(* Schneider Machine Expert - Basic project Grease Machine, file version 2.6.0.0 *)
(* ProjectInformations: Name=New project *)

HARDWARE
  Cpu 0: TM221CE40R
  EthernetConfiguration: NetworkName=M221, IpAllocationMode=FixedAddress, IpAddress=192.168.0.3, SubnetMask=255.255.255.0
  SerialLineConfiguration: Baud=Baud19200, Parity=ParityEven, DataBits=DataBits8, StopBits=StopBits1, PhysicalMedium=PhysicalMediumRs485, TransmissionMode=TransmissionModeModbusRtu, SlaveId=1, Addressing=SlaveAddressing
  MastTask: UsePeriodScanMode=false, PeriodScan=100
  FastTask: Period=255
  CpuBehavior: StartingMode=StartAsPreviousState, AutoSaveRamOnEeprom=true, WatchdogPeriod=250

SYMBOLS  (address, symbol, comment, settings)
  %M0         "RST HMI"
  %M1         "M_BTN START"
  %M2         "M_SENSOR CERTAIN"
  %M3         "M_SENSOR TABLE"
  %M4         "M_BTN CYCLE START"
  %M5         "M_EMG"
  %M6         "M_PROCESS DONE"
  %M7         "M_GREASE EMPTY"
  %M8         "M_GREASE TRIGGER"
  %M9         "M_Q GREASE ACTIVE"
  %M10        "M_Q CERTAIN SENSOR"
  %M11        "M_Q CYCLE START"
  %M12        "M_Q EMERGENCY"
  %M13        "M_Q RED LAMP"
  %M14        "M_Q YELLOW LAMP"
  %M15        "M_Q GREEN LAMP"
  %M16        "M_Q BUZZER"
  %M17        "RED LAMP 2"
  %M18        "TRIGGER YELLOW LAMP"
  %M19        "PAUSE"
  %M20        "FINISH RUN"
  %M21        "RESET BUZZER"
  %M22        "MEMORY M2"
  %M23        "M_TABLE_HMI"
  %M30        "M_START"
  %M31        "M_START HMI"
  %M32        "M_RUN_EMG"
  %M33        "TRIGER_ROBOT_HOME"
  %M34        "ROBOT_GO_HOME"
  %M47        "M_EMG"
  %M49        "POLARITY CHECKED"
  %M50        "NEGATIVE"
  %M51        "POSITIVE"
  %M52        "FIRST RUN"
  %M53        "DONE CUTTING"
  %M54        "NEGATIVE READY"
  %M55        "TRIGGER"
  %M56        "COUNTER OUTPUT"
  %M100       "START GUI"
  %M102       "M_START"
  %MW0        "Count Output"
  %I0.1       "BTN START"
  %I0.2       "SENSOR CERTAIN"
  %I0.3       "SENSOR TABLE"
  %I0.4       "BTN CYCLE START"
  %I0.5       "BTN EMG"
  %I0.6       "PROCESS DONE"
  %I0.7       "TANK EMPTY"
  %I0.8       "TRIGGER GREASE"
  %Q0.0       "GREASE ACTIVE"
  %Q0.1       "CERTAIN SENSOR"
  %Q0.2       "CYCLE START"
  %Q0.3       "EMERGENCY"
  %Q0.4       "RED_LAMP"
  %Q0.5       "YELLOW_LAMP"
  %Q0.6       "GREEN_LAMP"
  %Q0.7       "BUZZER"

POU New POU
  (* SectionNumber=1 *)

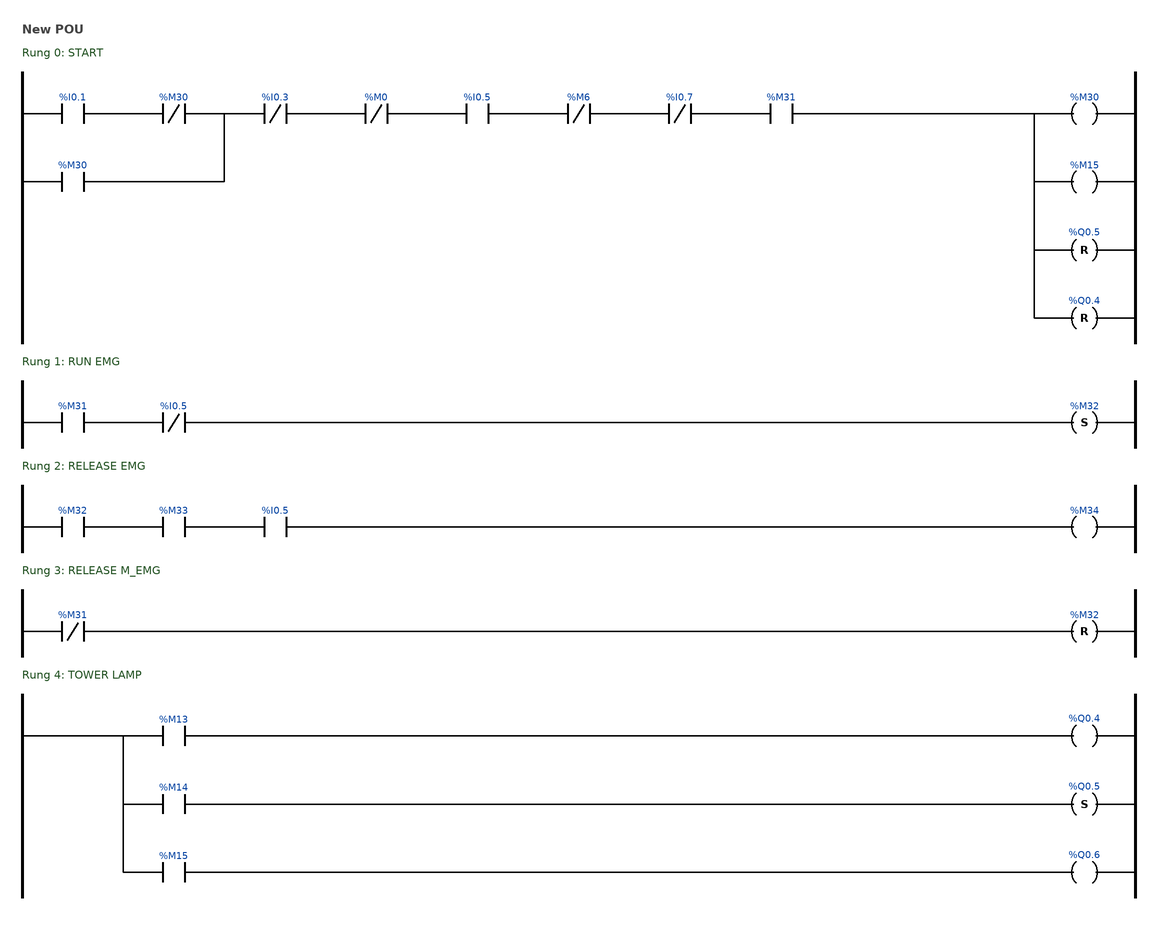

// Rung 0: START
  LD %I0.1
  ANDN %M30
  OR %M30
  ANDN %I0.3
  ANDN %M0
  AND %I0.5
  ANDN %M6
  ANDN %I0.7
  AND %M31
  ST %M30
  ST %M15
  R %Q0.5
  R %Q0.4
  // as ST:
  //   _t1 := (%I0.1 AND NOT %M30 OR %M30) AND NOT %I0.3 AND NOT %M0 AND %I0.5 AND NOT %M6 AND NOT %I0.7 AND %M31;
  //   %M30 := _t1;
  //   %M15 := _t1;
  //   IF _t1 THEN %Q0.5 := FALSE; END_IF;
  //   IF _t1 THEN %Q0.4 := FALSE; END_IF;

// Rung 1: RUN EMG
  LD %M31
  ANDN %I0.5
  S %M32
  // as ST:
  //   IF %M31 AND NOT %I0.5 THEN %M32 := TRUE; END_IF;

// Rung 2: RELEASE EMG
  LD %M32
  AND %M33
  AND %I0.5
  ST %M34
  // as ST:
  //   %M34 := %M32 AND %M33 AND %I0.5;

// Rung 3: RELEASE M_EMG
  LDN %M31
  R %M32
  // as ST:
  //   IF NOT %M31 THEN %M32 := FALSE; END_IF;

// Rung 4: TOWER LAMP
  LD 1
  MPS
  AND %M13
  ST %Q0.4
  MRD
  AND %M14
  S %Q0.5
  MPP
  AND %M15
  ST %Q0.6
  // as ST:
  //   %Q0.4 := %M13;
  //   IF %M14 THEN %Q0.5 := TRUE; END_IF;
  //   %Q0.6 := %M15;

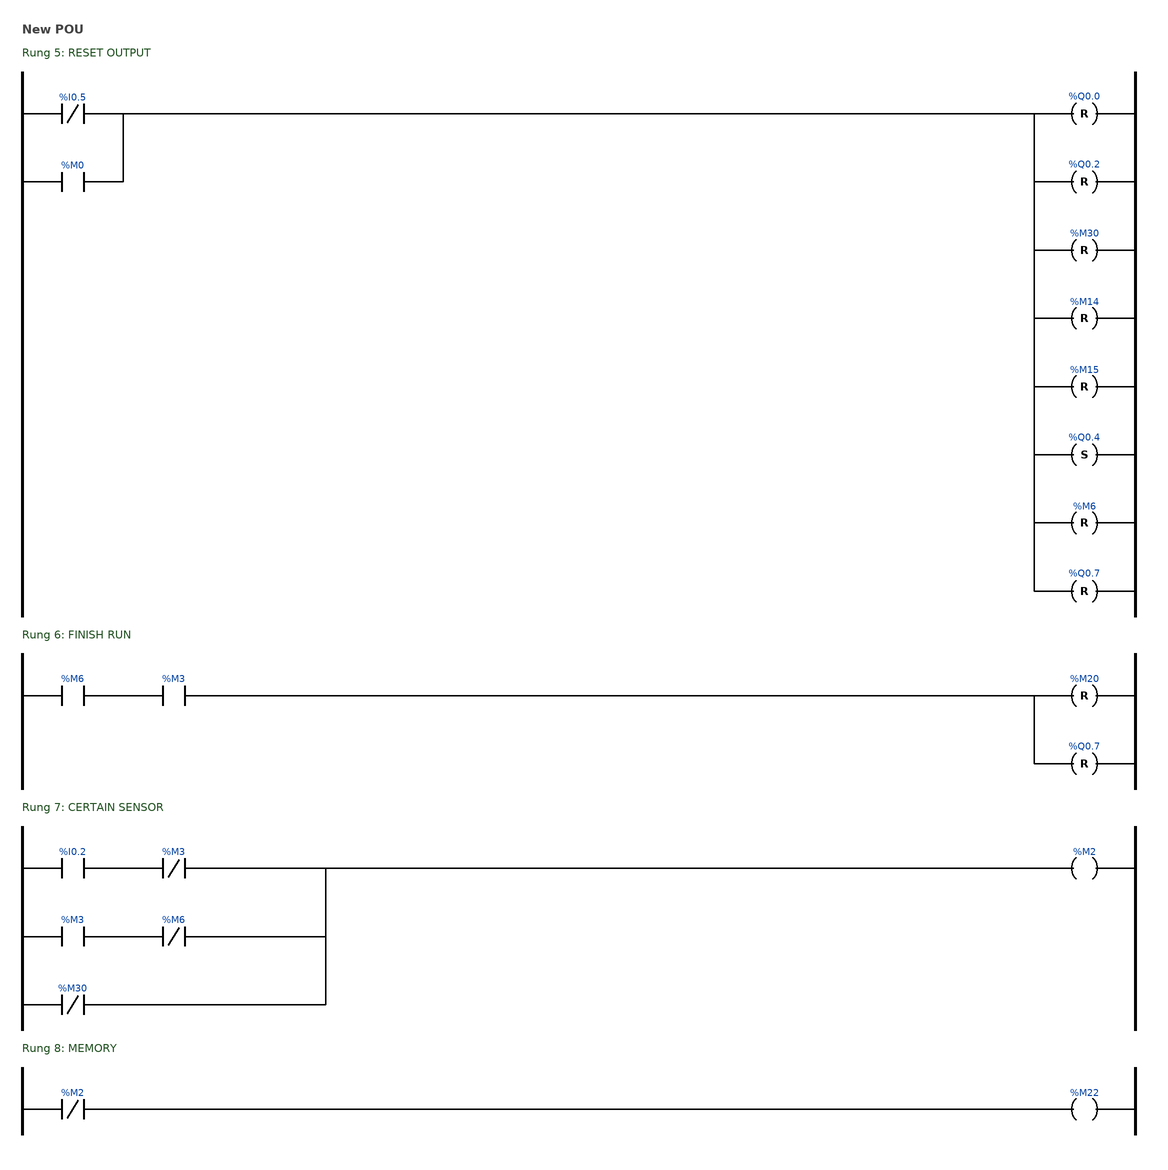

// Rung 5: RESET OUTPUT
  LDN %I0.5
  OR %M0
  R %Q0.0
  R %Q0.2
  R %M30
  R %M14
  R %M15
  S %Q0.4
  R %M6
  R %Q0.7
  // as ST:
  //   IF NOT %I0.5 OR %M0 THEN %Q0.0 := FALSE; END_IF;
  //   IF NOT %I0.5 OR %M0 THEN %Q0.2 := FALSE; END_IF;
  //   IF NOT %I0.5 OR %M0 THEN %M30 := FALSE; END_IF;
  //   IF NOT %I0.5 OR %M0 THEN %M14 := FALSE; END_IF;
  //   IF NOT %I0.5 OR %M0 THEN %M15 := FALSE; END_IF;
  //   IF NOT %I0.5 OR %M0 THEN %Q0.4 := TRUE; END_IF;
  //   IF NOT %I0.5 OR %M0 THEN %M6 := FALSE; END_IF;
  //   IF NOT %I0.5 OR %M0 THEN %Q0.7 := FALSE; END_IF;

// Rung 6: FINISH RUN
  LD %M6
  AND %M3
  R %M20
  R %Q0.7
  // as ST:
  //   IF %M6 AND %M3 THEN %M20 := FALSE; END_IF;
  //   IF %M6 AND %M3 THEN %Q0.7 := FALSE; END_IF;

// Rung 7: CERTAIN SENSOR
  LD %I0.2
  ANDN %M3
  OR( %M3
  ANDN %M6
  )
  ORN %M30
  ST %M2
  // as ST:
  //   %M2 := %I0.2 AND NOT %M3 OR %M3 AND NOT %M6 OR NOT %M30;

// Rung 8: MEMORY
  LDN %M2
  ST %M22
  // as ST:
  //   %M22 := NOT %M2;

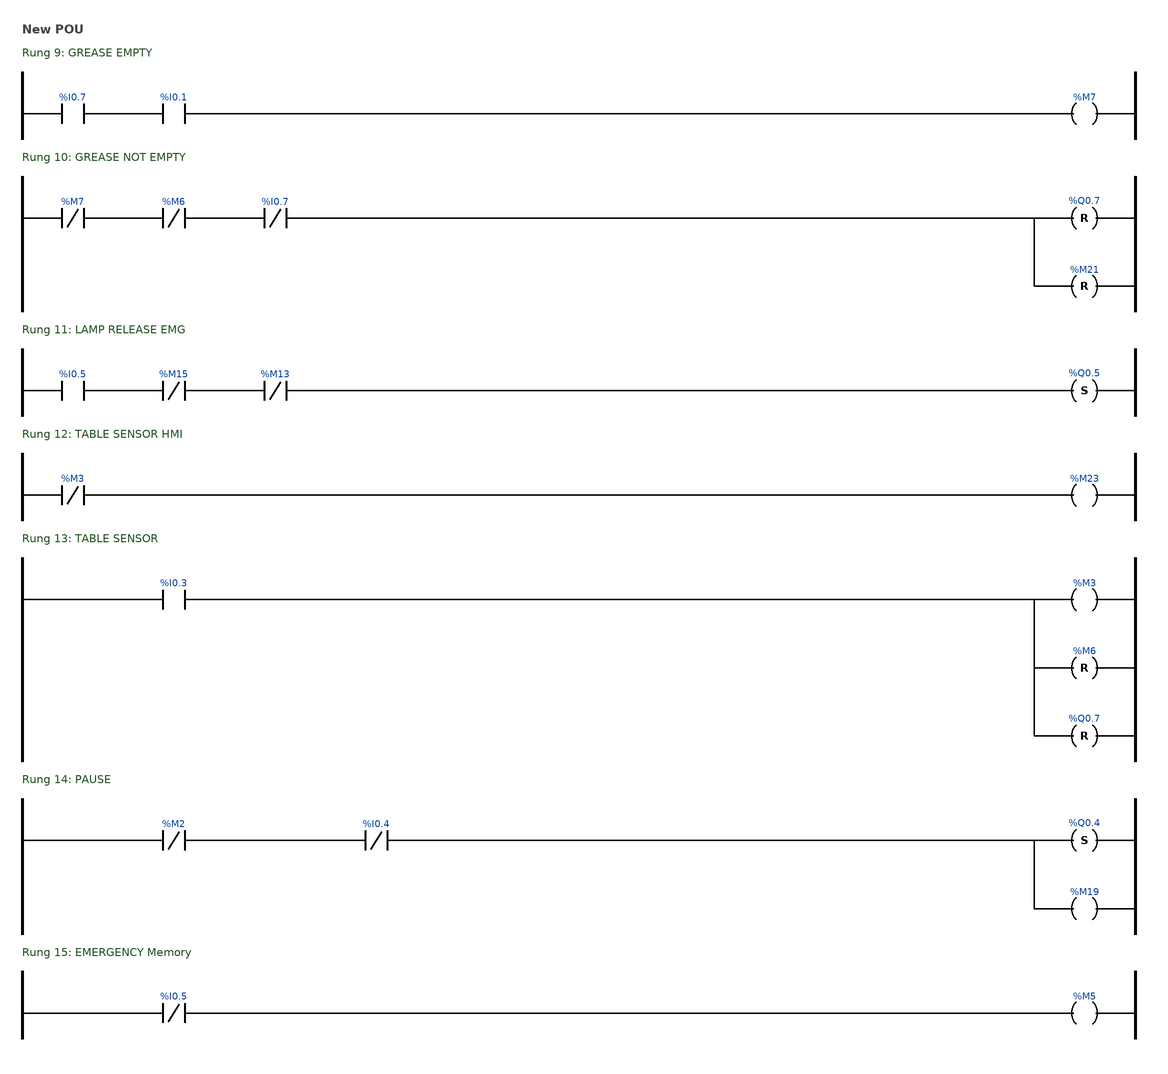

// Rung 9: GREASE EMPTY
  LD %I0.7
  AND %I0.1
  ST %M7
  // as ST:
  //   %M7 := %I0.7 AND %I0.1;

// Rung 10: GREASE NOT EMPTY
  LDN %M7
  ANDN %M6
  ANDN %I0.7
  R %Q0.7
  R %M21
  // as ST:
  //   IF NOT %M7 AND NOT %M6 AND NOT %I0.7 THEN %Q0.7 := FALSE; END_IF;
  //   IF NOT %M7 AND NOT %M6 AND NOT %I0.7 THEN %M21 := FALSE; END_IF;

// Rung 11: LAMP RELEASE EMG
  LD %I0.5
  ANDN %M15
  ANDN %M13
  S %Q0.5
  // as ST:
  //   IF %I0.5 AND NOT %M15 AND NOT %M13 THEN %Q0.5 := TRUE; END_IF;

// Rung 12: TABLE SENSOR HMI
  LDN %M3
  ST %M23
  // as ST:
  //   %M23 := NOT %M3;

// Rung 13: TABLE SENSOR
  LD %I0.3
  ST %M3
  R %M6
  R %Q0.7
  // as ST:
  //   %M3 := %I0.3;
  //   IF %I0.3 THEN %M6 := FALSE; END_IF;
  //   IF %I0.3 THEN %Q0.7 := FALSE; END_IF;

// Rung 14: PAUSE
  LDN %M2
  ANDN %I0.4
  S %Q0.4
  ST %M19
  // as ST:
  //   IF NOT %M2 AND NOT %I0.4 THEN %Q0.4 := TRUE; END_IF;
  //   %M19 := NOT %M2 AND NOT %I0.4;

// Rung 15: EMERGENCY Memory
  LDN %I0.5
  ST %M5
  // as ST:
  //   %M5 := NOT %I0.5;

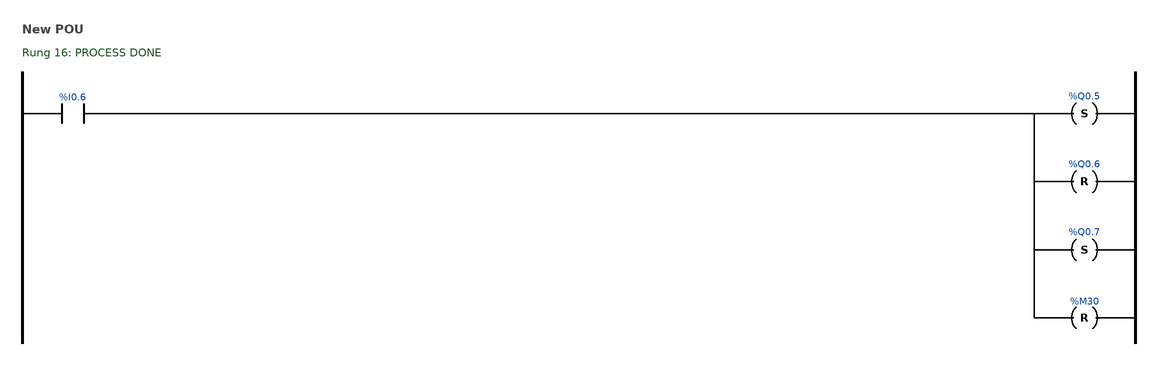

// Rung 16: PROCESS DONE
  LD %I0.6
  S %Q0.5
  R %Q0.6
  S %Q0.7
  R %M30
  // as ST:
  //   IF %I0.6 THEN %Q0.5 := TRUE; END_IF;
  //   IF %I0.6 THEN %Q0.6 := FALSE; END_IF;
  //   IF %I0.6 THEN %Q0.7 := TRUE; END_IF;
  //   IF %I0.6 THEN %M30 := FALSE; END_IF;

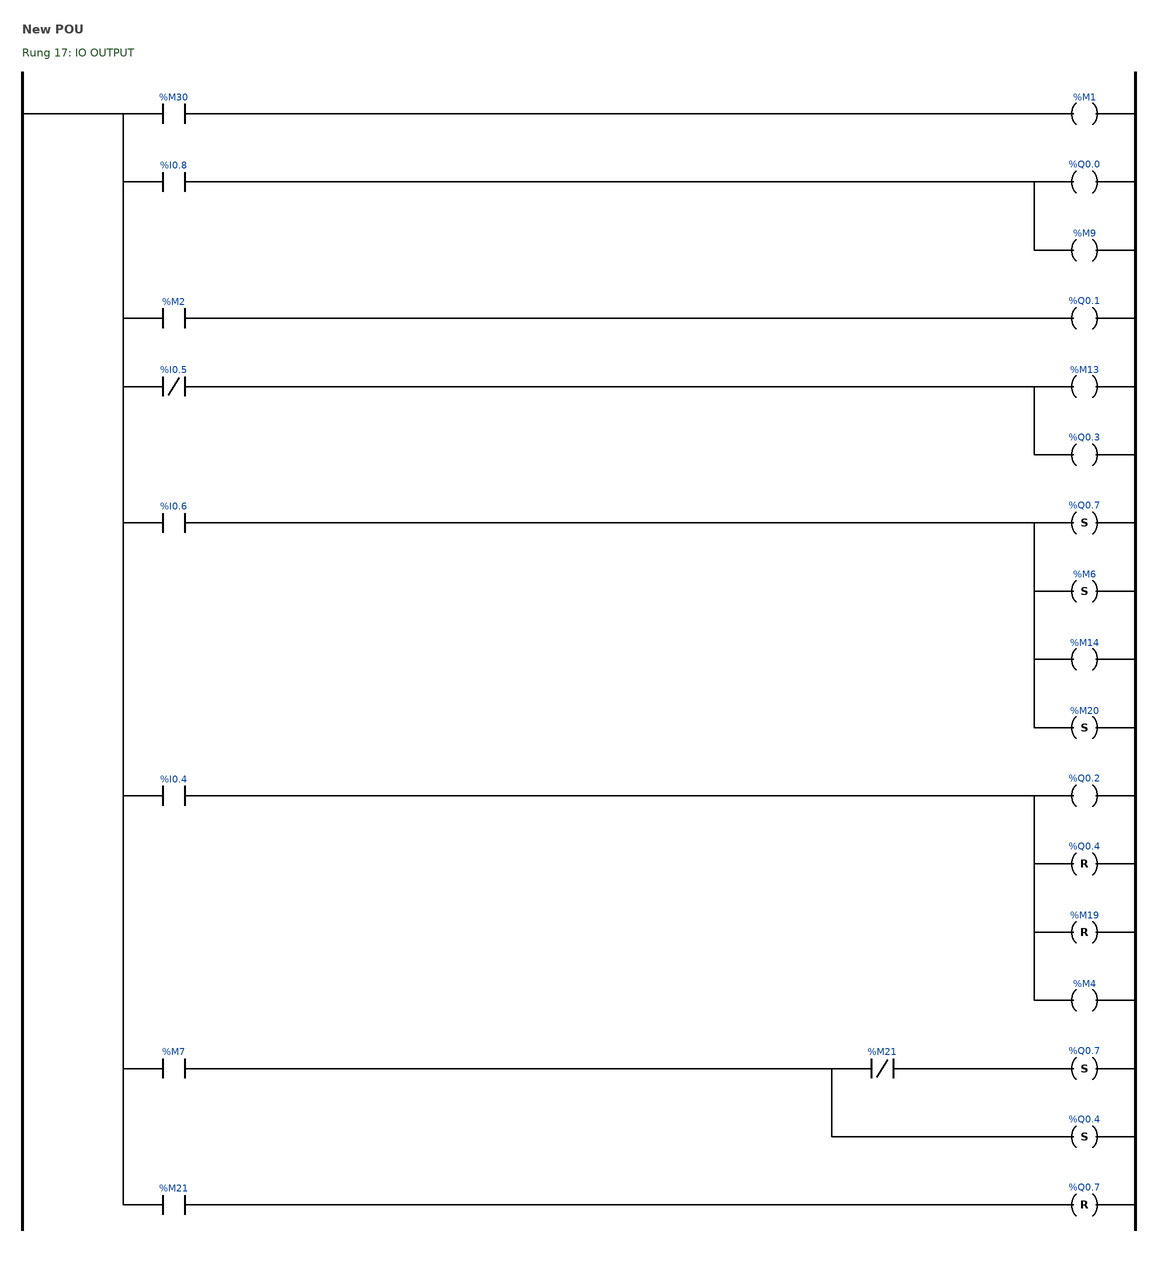

// Rung 17: IO OUTPUT
  LD 1
  MPS
  AND %M30
  ST %M1
  MRD
  AND %I0.8
  ST %Q0.0
  ST %M9
  MRD
  AND %M2
  ST %Q0.1
  MRD
  ANDN %I0.5
  ST %M13
  ST %Q0.3
  MRD
  AND %I0.6
  S %Q0.7
  S %M6
  ST %M14
  S %M20
  MRD
  AND %I0.4
  ST %Q0.2
  R %Q0.4
  R %M19
  ST %M4
  MRD
  AND %M7
  MPS
  ANDN %M21
  S %Q0.7
  MPP
  S %Q0.4
  MPP
  AND %M21
  R %Q0.7
  // as ST:
  //   %M1 := %M30;
  //   %Q0.0 := %I0.8;
  //   %M9 := %I0.8;
  //   %Q0.1 := %M2;
  //   %M13 := NOT %I0.5;
  //   %Q0.3 := NOT %I0.5;
  //   IF %I0.6 THEN %Q0.7 := TRUE; END_IF;
  //   IF %I0.6 THEN %M6 := TRUE; END_IF;
  //   %M14 := %I0.6;
  //   IF %I0.6 THEN %M20 := TRUE; END_IF;
  //   %Q0.2 := %I0.4;
  //   IF %I0.4 THEN %Q0.4 := FALSE; END_IF;
  //   IF %I0.4 THEN %M19 := FALSE; END_IF;
  //   %M4 := %I0.4;
  //   IF %M7 AND NOT %M21 THEN %Q0.7 := TRUE; END_IF;
  //   IF %M7 THEN %Q0.4 := TRUE; END_IF;
  //   IF %M21 THEN %Q0.7 := FALSE; END_IF;
